FUNCTION_BLOCK PUBLIC IB_StopRobotClearStation
VAR_INPUT
END_VAR
VAR_OUTPUT
END_VAR
VAR
	xTrigger :BOOL := FALSE; // triggers processing
	State : eIB_StopRobotClearStaState := eIB_StopRobotClearStaState.eUnknown;
	NextState : eIB_StopRobotClearStaState := eIB_StopRobotClearStaState.eUnknown;
	bFirst : BOOL := TRUE;
	VUT : BYTE; //VehicleID Under Station
	DwellTimer : TON;
END_VAR

CASE State OF
eIB_StopRobotClearStaState.eUnknown:
	NextState := eIB_StopRobotClearStaState.eReady;
	
eIB_StopRobotClearStaState.eInit:

eIB_StopRobotClearStaState.eHoming:

eIB_StopRobotClearStaState.eReady:
	IF (xTrigger) THEN
		NextState := eIB_StopRobotClearStaState.eProcessing;		
		DwellTimer(IN:=FALSE);
	END_IF

eIB_StopRobotClearStaState.eDwell:	

eIB_StopRobotClearStaState.eProcessing:
	IF(Stations.fbLoad1Sta.HoldVehicle_IBStop = FALSE) THEN
		NextState := eIB_StopRobotClearStaState.eDepart;
	END_IF

eIB_StopRobotClearStaState.eDepart:
		Stations.fbRoutePlanner.M_NotifyVehStaCmpl(StationIndex:= MM_CONST.IB_STOP_ROBOT_CLEAR_STA, VehicleID := VUT);
		xTrigger := FALSE;
		IF (Stations.fbCycleControl.StopRequested) THEN
			NextState := eIB_StopRobotClearStaState.eStopActive;
		ELSE
			NextState := eIB_StopRobotClearStaState.eReady;		
		END_IF
		
eIB_StopRobotClearStaState.eStopActive:
	IF (NOT Stations.fbCycleControl.StopRequested) THEN
		NextState := eIB_StopRobotClearStaState.eReady;	
	END_IF
		
eIB_StopRobotClearStaState.eError:
END_CASE

IF (State <> NextState) THEN
	bFirst := TRUE;
ELSE
	bFirst := FALSE;
END_IF

State := NextState;
//Status.StationsState[MM_CONST.IB_STOP_ROBOT_CLEAR_STA_HMI_STATE] := State;
//AssignStationStatusForHMI();

METHOD PUBLIC ClearVehicleTrigger : BOOL
VAR_INPUT
END_VAR
xTrigger := FALSE;
State  := eIB_StopRobotClearStaState.eUnknown;
NextState  := eIB_StopRobotClearStaState.eUnknown;
bFirst  := TRUE;
END_METHOD

PROPERTY PUBLIC Trigger : BOOL
SET
xTrigger := Trigger;
END_SET
END_PROPERTY

PROPERTY PUBLIC VehicleUnderTest : BYTE
GET
VehicleUnderTest := VUT;
END_GET
SET
VUT := VehicleUnderTest;
END_SET
END_PROPERTY

END_FUNCTION_BLOCK

(* stored: Version 1.1.0.1, ProductVersion 3.1.4020.12
   POU IB_StopRobotClearStation: Id {4d0c533c-d737-41da-aadf-236b1de6a77c}, SpecialFunc None
   Method ClearVehicleTrigger: Id {d31806d1-389e-4abb-b8ff-d2fb476700f0}
   Property Trigger: Id {40d14ebd-90f9-4db6-89df-0f4886d7b4b1}
   Set Set: Id {86465deb-a801-4269-bf98-4c153f17f580}
   Property VehicleUnderTest: Id {cb55f436-0b0b-4803-a6c4-9a942dad1487}
   Get Get: Id {0f451fc6-5c3d-4585-9138-09baf63b0899}
   Set Set: Id {d2921964-018f-4f5f-b0d8-94969bcb7406} *)
